TYPE "Type_IO"
VERSION : 0.1
   STRUCT
      Ind : Int := -1;
      Stato : Int;
      BVal : Bool;
      IVal : Int;
      DVal : DInt;
      RVal : Real;
      "FC" : Real;
      Offset : Real;
      BProgVal : Bool;
      DProgVal : DInt;
   END_STRUCT;

END_TYPE

